{attribute 'qualified_only'}
{attribute 'strict'}
TYPE E_StartVisu :
(
	Logo := 0,
	Settings,
	Parameter,
	Manual,
	SemiAutomatic,
	Automatic
)DINT;
END_TYPE

(* stored: Version 1.1.0.1, ProductVersion 3.1.4024.5
   EnumerationTextList E_StartVisu: Id {f72244d6-971b-4c1b-8ca1-7c82c03cdf0f} *)
